PROGRAM Axis04_Manual
VAR
	Always_ON	:	BOOL	:=TRUE	;//상시 ON 
	Always_OFF	:	BOOL	:=FALSE	;//상시 OFF
END_VAR

// NETWORK 1

END_PROGRAM

(* stored: Version 1.1.0.1, ProductVersion 3.1.4024.15
   POU Axis04_Manual: Id {0bc47764-b7c2-4f2e-b58d-d775da31f11d}, SpecialFunc None *)
